// TIA Portal V20 export
TYPE "LBP_typeModularMcpLedAttribute"
TITLE = Modular MCP image / Image MCP modulaire
// User data type for LBP_typeModularMcpKeypadRecord (sub type) / Type de données utilisateur pour LBP_typeModularMcpKeypadRecord (sous-type)
   STRUCT
      keyIndex : USInt;   // index of key / indice de touche
      red : USInt;   // intensity of red LED / intensité de la LED rouge
      green : USInt;   // intensity of green LED / intensité de la LED verte
      blue : USInt;   // intensity of blue LED / intensité de la LED bleue
   END_STRUCT;
END_TYPE
